FUNCTION F_StringToWstringPL : WSTRING
VAR_INPUT
	sInput	: STRING;
END_VAR
VAR
	iNum			: INT;	
//	iChar			: INT;
	iLen			: INT;
END_VAR

iLen	:=LEN(sInput);	//ilość znaków w stringu
FOR iNum:=0 TO iLen-1 DO
	CASE sInput[iNum] OF
		
		140://Ś
			F_StringToWstringPL[iNum]	:= 90+256;
		143://Ź
			F_StringToWstringPL[iNum]	:= 121+256;	
		156://ś
			F_StringToWstringPL[iNum]	:= 91+256;
		159://ź
			F_StringToWstringPL[iNum]	:= 122+256;
		163://Ł
			F_StringToWstringPL[iNum]	:= 65+256;
		165://Ą
			F_StringToWstringPL[iNum]	:= 4+256;
		175://Ż
			F_StringToWstringPL[iNum]	:= 123+256;
		179://ł
			F_StringToWstringPL[iNum]	:= 66+256;
		185://ą
			F_StringToWstringPL[iNum]	:= 5+256;
		191://ż
			F_StringToWstringPL[iNum]	:= 124+256;
		198://Ć
			F_StringToWstringPL[iNum]	:= 6+256;
		202://Ę
			F_StringToWstringPL[iNum]	:= 24+256;	
		209://Ń
			F_StringToWstringPL[iNum]	:= 67+256;
//		211://Ó - bez zmiany
		230://ć
			F_StringToWstringPL[iNum]	:= 7+256;
		234://ę
			F_StringToWstringPL[iNum]	:= 25+256;
		241://ń
			F_StringToWstringPL[iNum]	:= 68+256;

//		243://ó - bez zmiany
		
		ELSE
			F_StringToWstringPL[iNum]	:= sInput[iNum];
	END_CASE

END_FOR
F_StringToWstringPL[iLen]:= 0;//Dodane 0 - koniec wstringa



//F_StringToWstringPL:="";

//FOR iNum:=1 TO LEN(sInput) DO
//	iChar	:= F_ToASC(MID(sInput,1,iNum));
//	CASE iChar OF
//		140:
//			F_StringToWstringPL	:= WCONCAT(F_StringToWstringPL,"Ś");
//		143:
//			F_StringToWstringPL	:= WCONCAT(F_StringToWstringPL,"Ź");
//		156:
//			F_StringToWstringPL	:= WCONCAT(F_StringToWstringPL,"ś");
//		159:
//			F_StringToWstringPL	:= WCONCAT(F_StringToWstringPL,"ź");
//		163:
//			F_StringToWstringPL	:= WCONCAT(F_StringToWstringPL,"Ł");
//		165:
//			F_StringToWstringPL	:= WCONCAT(F_StringToWstringPL,"Ą");
//		175:
//			F_StringToWstringPL	:= WCONCAT(F_StringToWstringPL,"Ż");	
//		179:
//			F_StringToWstringPL	:= WCONCAT(F_StringToWstringPL,"ł");
//		185:
//			F_StringToWstringPL	:= WCONCAT(F_StringToWstringPL,"ą");
//		191:
//			F_StringToWstringPL	:= WCONCAT(F_StringToWstringPL,"ż");
//		198:
//			F_StringToWstringPL	:= WCONCAT(F_StringToWstringPL,"Ć");
//		202:
//			F_StringToWstringPL	:= WCONCAT(F_StringToWstringPL,"Ę");		
//		209:
//			F_StringToWstringPL	:= WCONCAT(F_StringToWstringPL,"Ń");
//		211:
//			F_StringToWstringPL	:= WCONCAT(F_StringToWstringPL,"Ó");
//		230:
//			F_StringToWstringPL	:= WCONCAT(F_StringToWstringPL,"ć");
//		234:
//			F_StringToWstringPL	:= WCONCAT(F_StringToWstringPL,"ę");
//		241:
//			F_StringToWstringPL	:= WCONCAT(F_StringToWstringPL,"ń");
//		243:
//			F_StringToWstringPL	:= WCONCAT(F_StringToWstringPL,"ó");

		
//		ELSE
//			F_StringToWstringPL	:= WCONCAT(F_StringToWstringPL,TO_WSTRING(MID(sInput,1,iNum)));
			
//	END_CASE
//END_FOR

END_FUNCTION

(* stored: Version 1.1.0.1, ProductVersion 3.1.4026.13, FileIdentifier 4d60ceb282a9d0926e4f8309c3465d01533c1473, FileSignature 7268ced2260da5a3635f807717e248c8136623d7acb5b571c0ff46c8ccbe1ff6afa62f83e04be1efa0b968d9dd39741dabbcdfa0c6777ea687fd5cabf98bd7f3fec40531b0cc9be4ad3358a0594acd930a3de0424f2b8970ed3afdfa30c710ab827487ac0cc4410563217652c15ed729afea28961ed02599e54adaee0b754aeed5f6b3e86be950b888c3a40d6d8454beea276baa56b3e96ebbdd15efc14479c7ecfbe70e8c2beeda4d0cbcca48b0fe7f03aae9250281960545f44b67698e04fe98495d49c4bd0efa1dbc8957d8c1b0557570fea3a591288c22c99144f5d7e94192778b6d97aed8cafc7b7f108a1ec6d20153238b1a44f81570a18e442a4f4e49
   POU F_StringToWstringPL: Id {660c2fb8-f49b-4230-871d-cf45f7d27505}, SpecialFunc None *)
